SUBAPPLICATION AuxInput_Heckschieber_UP (* Subapplication Type *)
  (* Standard: 61499-2 *)
  (* Version 1.0, 2023-02-11, franz *)
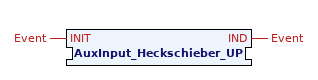
  EVENT_INPUT
    INIT;
  END_EVENT
  EVENT_OUTPUT
    IND;
  END_EVENT
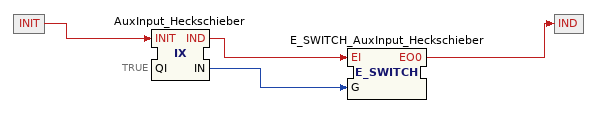
  FBS
    E_SWITCH_AuxInput_Heckschieber : E_SWITCH;
    AuxInput_Heckschieber : IX(QI := TRUE);
  END_FBS
  EVENT_CONNECTIONS
    AuxInput_Heckschieber.IND TO E_SWITCH_AuxInput_Heckschieber.EI;
    INIT TO AuxInput_Heckschieber.INIT;
    E_SWITCH_AuxInput_Heckschieber.EO0 TO IND;
  END_CONNECTIONS
  DATA_CONNECTIONS
    AuxInput_Heckschieber.IN TO E_SWITCH_AuxInput_Heckschieber.G;
  END_CONNECTIONS
END_SUBAPPLICATION
